Fanuc KAREL source: mth_abs.kl

PROGRAM mth_abs
%NOBUSYLAMP
%NOLOCKGROUP

VAR
	out_reg : INTEGER
	val : REAL
%from tpe.klh %import get_real_arg,get_int_arg
%from registers.klh %import set_real
%from math.builtins.klh %import abs

BEGIN
	val = tpe__get_real_arg(1)
	out_reg = tpe__get_int_arg(2)
	registers__set_real(out_reg, math__abs(val))
END mth_abs
